Staubli VAL3: TestSuccionar.dtx

mdesc mNomSpeed
jointRx JApproach1 = {j1=-7.51945495605469, j2=-3.64574456214905, j3=61.4223289489746, j5=122.22339630127, j6=172.480560302734}
jointRx jGetCinta = {j1=-61.1670760931322, j2=47.4709417128017, j3=73.8913906677858, j4=0.557661040069446, j5=59.5118412194821, j6=118.546320517872}
pointRx pApprBins = {x=391.677002218024, y=-12.0780241054472, z=88.9240908929814, rx=-179.99999141576, ry=8.18584317852812E-07, rz=5.54303290954861E-07, fatherId=world[0]}
tool tToolSuccion = {z=110, fatherId=flange[0], ioLink=valve1}
